FUNCTION_BLOCK Test_RaiseNotification_UpdatesNotificationHandler EXTENDS tcl_SimpleUnitTestLibrary.T_UnitTestBase
VAR
    Source  : T_Notification;
    Handler : T_NotificationHandler;
    
    ResultString : T_MaxString;
END_VAR

Handler.FB_init(
    bInitRetains := FALSE,  
    bInCopyCode  := FALSE);

Source.ClearNotificationHandlers();
Source.AddNotificationHandler(Handler);

Source.Args.Clear().Add_STRING('Big long string passed to the notification handler for later use');
Source.Raise();

Assertion.AssertEquals_BOOL(
    Expected     := TRUE,
    Actual       := Handler.IsRaised(),
    VariableName := 'Handler.IsRaised()');
    
ResultString := Handler.NotificationArgs.Read_STRING();

Assertion.AssertEquals_STRING(
    Expected     := 'Big long string passed to the notification handler for later use',
    Actual       := ResultString,
    VariableName := 'ResultString');
    
    

TestFinished();

END_FUNCTION_BLOCK

(* stored: Version 1.1.0.1, ProductVersion 3.1.4024.4
   POU Test_RaiseNotification_UpdatesNotificationHandler: Id {4e551fab-9c56-45bf-b8fd-d0a5797af32e}, SpecialFunc None *)
